// TIA Portal project "projet sadokkkkkkalasou" (V16)
// Vorlageprojekt für das Buch mit Zielsystem S7-1200

(* hardware
DEVICE "S7-1200-Station_1"  S7-1200 Station
   slot 0: "Baugruppenträger_0"  Rack  V1.0
   slot 1: "PLC_1"  CPU 1211C DC/DC/DC  6ES7 211-1AE40-0XB0  V4.1
*)

// ===== PLC "PLC_1"  CPU 1211C DC/DC/DC =====

VAR_GLOBAL   // PLC tag table "Standard-Variablentabelle"
   "km1" AT %Q0.0 : Bool;
   "km2" AT %Q0.2 : Bool;
   "GRAB" AT %Q0.1 : Bool;
   "MOVE X" AT %Q0.3 : Bool;
   "MOVE Z" AT %Q0.4 : Bool;
   "PUSHER" AT %Q0.5 : Bool;
   "LH" AT %I0.1 : Bool;
   "LL" AT %I0.2 : Bool;
   "CP" AT %I0.3 : Bool;
   "CC" AT %I0.4 : Bool;
   "PD" AT %I0.5 : Bool;
   "SZ" AT %I0.6 : Bool;
   "SX" AT %I0.7 : Bool;
   "START" AT %I1.0 : Bool;
   "Moving X" AT %I1.1 : Bool;
   "moving Z" AT %I1.2 : Bool;
   "DS4" AT %I1.3 : Bool;
   "STOP" AT %I1.4 : Bool;
   "km3" AT %Q1.5 : Bool;
   "FC2" AT %I1.6 : Bool;
   "FC1" AT %I1.7 : Bool;
   "Emiteur1" AT %Q2.0 : Bool;
   "Emiteur2" AT %Q2.1 : Bool;
   "Rb1" AT %Q2.2 : Bool;
   "Rb2" AT %Q2.3 : Bool;
   "rs1" AT %I2.4 : Bool;
   "rs2" AT %I2.5 : Bool;
   "cc2" AT %I3.1 : Bool;
   "sz2" AT %I3.2 : Bool;
   "sx2" AT %I3.3 : Bool;
   "rotccw" AT %Q2.4 : Bool;
   "rotcw" AT %Q2.5 : Bool;
   "rot1" AT %I3.4 : Bool;
   "rot4" AT %I2.7 : Bool;
   "km4" AT %Q2.7 : Bool;
   "FC3" AT %I3.0 : Bool;
   "Emiteur3" AT %Q0.6 : Bool;
   "rb3" AT %Q0.7 : Bool;
   "rb31" AT %Q1.0 : Bool;
   "rb32" AT %Q1.1 : Bool;
   "rb11" AT %Q1.2 : Bool;
   "rb21" AT %Q1.3 : Bool;
   "rb22" AT %Q1.4 : Bool;
   "red light" AT %Q1.6 : Bool;
   "green light" AT %Q1.7 : Bool;
   "yellow light" AT %Q2.6 : Bool;
END_VAR

// folder: System blocks/Program resources

DATA_BLOCK "IEC_Timer_0_DB"   // DB1
{ S7_Optimized_Access := 'TRUE' }
AUTHOR : Simatic
FAMILY : IEC
NAME : IEC_TMR
VERSION : 1.0
// stored: InstanceOfName IEC_TIMER
"IEC_TIMER"
BEGIN
END_DATA_BLOCK

DATA_BLOCK "IEC_Timer_0_DB_1"   // DB2
{ S7_Optimized_Access := 'TRUE' }
AUTHOR : Simatic
FAMILY : IEC
NAME : IEC_TMR
VERSION : 1.0
// stored: InstanceOfName IEC_TIMER
"IEC_TIMER"
BEGIN
END_DATA_BLOCK

DATA_BLOCK "IEC_Timer_0_DB_2"   // DB3
{ S7_Optimized_Access := 'TRUE' }
AUTHOR : Simatic
FAMILY : IEC
NAME : IEC_TMR
VERSION : 1.0
// stored: InstanceOfName IEC_TIMER
"IEC_TIMER"
BEGIN
END_DATA_BLOCK

DATA_BLOCK "IEC_Timer_0_DB_3"   // DB4
{ S7_Optimized_Access := 'TRUE' }
AUTHOR : Simatic
FAMILY : IEC
NAME : IEC_TMR
VERSION : 1.0
// stored: InstanceOfName IEC_TIMER
"IEC_TIMER"
BEGIN
END_DATA_BLOCK

DATA_BLOCK "IEC_Timer_0_DB_4"   // DB5
{ S7_Optimized_Access := 'TRUE' }
AUTHOR : Simatic
FAMILY : IEC
NAME : IEC_TMR
VERSION : 1.0
// stored: InstanceOfName IEC_TIMER
"IEC_TIMER"
BEGIN
END_DATA_BLOCK

DATA_BLOCK "IEC_Timer_0_DB_5"   // DB6
{ S7_Optimized_Access := 'TRUE' }
AUTHOR : Simatic
FAMILY : IEC
NAME : IEC_TMR
VERSION : 1.0
// stored: InstanceOfName IEC_TIMER
"IEC_TIMER"
BEGIN
END_DATA_BLOCK

DATA_BLOCK "IEC_Timer_0_DB_8"   // DB7
{ S7_Optimized_Access := 'TRUE' }
AUTHOR : Simatic
FAMILY : IEC
NAME : IEC_TMR
VERSION : 1.0
// stored: InstanceOfName IEC_TIMER
"IEC_TIMER"
BEGIN
END_DATA_BLOCK

DATA_BLOCK "IEC_Timer_0_DB_6"   // DB8
{ S7_Optimized_Access := 'TRUE' }
AUTHOR : Simatic
FAMILY : IEC
NAME : IEC_TMR
VERSION : 1.0
// stored: InstanceOfName IEC_TIMER
"IEC_TIMER"
BEGIN
END_DATA_BLOCK

DATA_BLOCK "IEC_Timer_0_DB_7"   // DB9
{ S7_Optimized_Access := 'TRUE' }
AUTHOR : Simatic
FAMILY : IEC
NAME : IEC_TMR
VERSION : 1.0
// stored: InstanceOfName IEC_TIMER
"IEC_TIMER"
BEGIN
END_DATA_BLOCK

DATA_BLOCK "IEC_Timer_0_DB_9"   // DB10
{ S7_Optimized_Access := 'TRUE' }
AUTHOR : Simatic
FAMILY : IEC
NAME : IEC_TMR
VERSION : 1.0
// stored: InstanceOfName IEC_TIMER
"IEC_TIMER"
BEGIN
END_DATA_BLOCK

DATA_BLOCK "IEC_Timer_0_DB_11"   // DB12
{ S7_Optimized_Access := 'TRUE' }
AUTHOR : Simatic
FAMILY : IEC
NAME : IEC_TMR
VERSION : 1.0
// stored: InstanceOfName IEC_TIMER
"IEC_TIMER"
BEGIN
END_DATA_BLOCK

DATA_BLOCK "IEC_Timer_0_DB_12"   // DB13
{ S7_Optimized_Access := 'TRUE' }
AUTHOR : Simatic
FAMILY : IEC
NAME : IEC_TMR
VERSION : 1.0
// stored: InstanceOfName IEC_TIMER
"IEC_TIMER"
BEGIN
END_DATA_BLOCK

// folder: (top level)

FUNCTION "MHJ-PLC-Lab-Function-S71200" : Void   // FC9000, SCL
{ S7_Optimized_Access := 'TRUE' }
VERSION : 0.1
   VAR_TEMP
      rdTimeReturn : Int;
      outputTime : DTL;
      SyncVal : Byte;
      forVal : Int;
      forVal_2 : Int;
      Value : Byte;
   END_VAR
   VAR CONSTANT
      CompVal : Byte := 16#34;
      Value_01 : Byte := 16#11;
      Value_01_DW : DWord := 16#A165_D992;
      Value_02_DW : DWord := 16#58BE_4401;
   END_VAR
BEGIN

   #Value:=PEEK(area := 16#82,
        dbNumber := 0,
        byteOffset := 511);
   #Value := #Value + 1;

   POKE(area := 16#82,
        dbNumber := 0,
        byteOffset := 511,
        value := #Value);

   POKE(area:=16#81,
        dbNumber:=0,
        byteOffset:=1016,
        value:=#Value_01_DW);
   POKE(area := 16#81,
        dbNumber := 0,
        byteOffset := 1020,
        value := #Value_02_DW);

   POKE(area := 16#81,
        dbNumber := 0,
        byteOffset := 511,
        value := B#16#00);

   FOR #forVal := 0 TO 120 DO
       FOR #forVal_2:=0 TO 10 DO
           #rdTimeReturn:=RD_SYS_T(#outputTime);
           #rdTimeReturn := WR_SYS_T(#outputTime);
           #rdTimeReturn := RD_SYS_T(#outputTime);
           #rdTimeReturn := WR_SYS_T(#outputTime);
       END_FOR;
       #SyncVal:= PEEK(area := 16#81,
                      dbNumber := 0,
                      byteOffset := 511);
       IF #SyncVal = #CompVal THEN
          GOTO M_1;
       END_IF;
   END_FOR;
   RETURN;

   M_1:
   POKE(area := 16#81,
        dbNumber := 0,
        byteOffset := 511,
        value := B#16#0);
END_FUNCTION

ORGANIZATION_BLOCK "Main"   // OB1, LAD, ProgramCycle
TITLE = "Main Program Sweep (Cycle)"
{ S7_Optimized_Access := 'TRUE' }
VERSION : 0.1
   VAR_INPUT
      Initial_Call : Bool;   // Initial call of this OB
      Remanence : Bool;   // =True, if remanent data are available
   END_VAR
   VAR_TEMP   // added for the SCL form of the ladder/FBD networks
      _w1 : Bool;
   END_VAR
BEGIN

REGION Network 1: Konnektierungsbaustein für PLC-Lab / liaison
   // Im Netzwerk 1 wird der Konnektierungsbaustein für PLC-Lab aufgerufen.
   // Dieser Aufruf darf nicht entfernt werden!
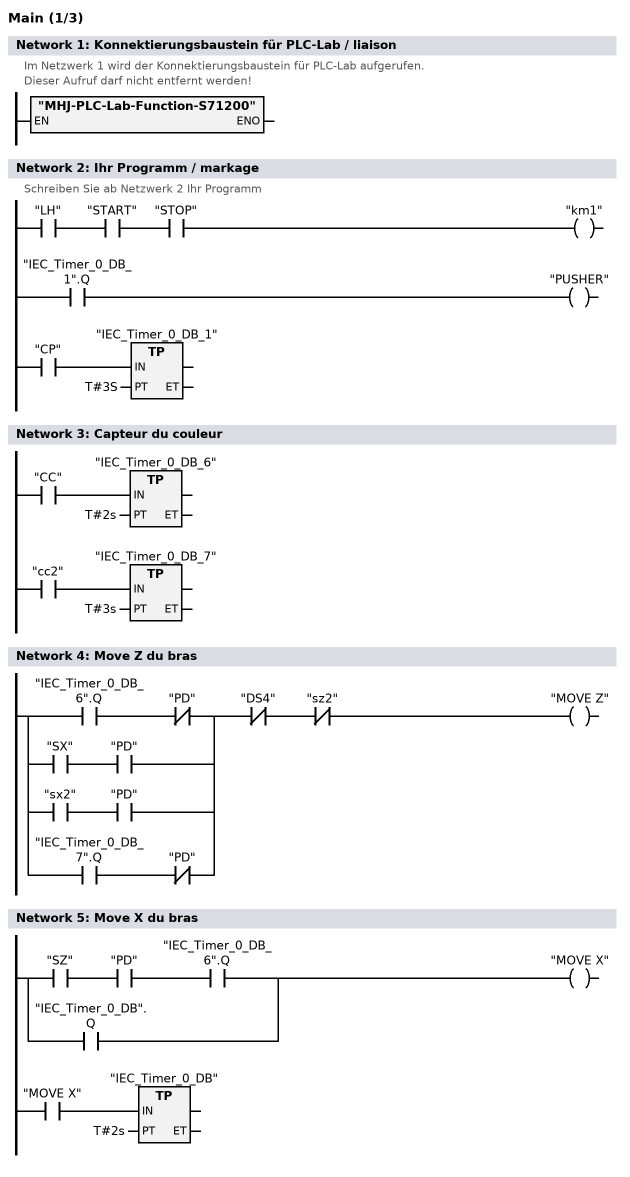
   RUNG wire#powerrail
      "MHJ-PLC-Lab-Function-S71200"()
   END_RUNG
   // the same network as SCL:
   "MHJ-PLC-Lab-Function-S71200"();
END_REGION

REGION Network 2: Ihr Programm / markage
   // Schreiben Sie ab Netzwerk 2 Ihr Programm
   "km1" := "LH" AND "START" AND "STOP";
   "PUSHER" := "IEC_Timer_0_DB_1".Q;
   "IEC_Timer_0_DB_1".TP(IN := "CP", PT := T#3S);
END_REGION

REGION Network 3: Capteur du couleur
   "IEC_Timer_0_DB_6".TP(IN := "CC", PT := T#2s);
   "IEC_Timer_0_DB_7".TP(IN := "cc2", PT := T#3s);
END_REGION

REGION Network 4: Move Z du bras
   RUNG wire#powerrail
      Contact( "IEC_Timer_0_DB_6".Q )
      I_Contact( "PD" )
      wire#w1
      I_Contact( "DS4" )
      I_Contact( "sz2" )
      Coil( "MOVE Z" )
   END_RUNG
   RUNG wire#powerrail
      Contact( "SX" )
      Contact( "PD" )
   END_RUNG wire#w1
   RUNG wire#powerrail
      Contact( "sx2" )
      Contact( "PD" )
   END_RUNG wire#w1
   RUNG wire#powerrail
      Contact( "IEC_Timer_0_DB_7".Q )
      I_Contact( "PD" )
   END_RUNG wire#w1
   // the same network as SCL:
   "MOVE Z" := (("IEC_Timer_0_DB_6".Q AND NOT "PD") OR ("SX" AND "PD") OR ("sx2" AND "PD") OR ("IEC_Timer_0_DB_7".Q AND NOT "PD")) AND NOT "DS4" AND NOT "sz2";
END_REGION

REGION Network 5: Move X du bras
   "MOVE X" := ("SZ" AND "PD" AND "IEC_Timer_0_DB_6".Q) OR "IEC_Timer_0_DB".Q;
   "IEC_Timer_0_DB".TP(IN := "MOVE X", PT := T#2s);
END_REGION

REGION Network 6: Rotation du bras
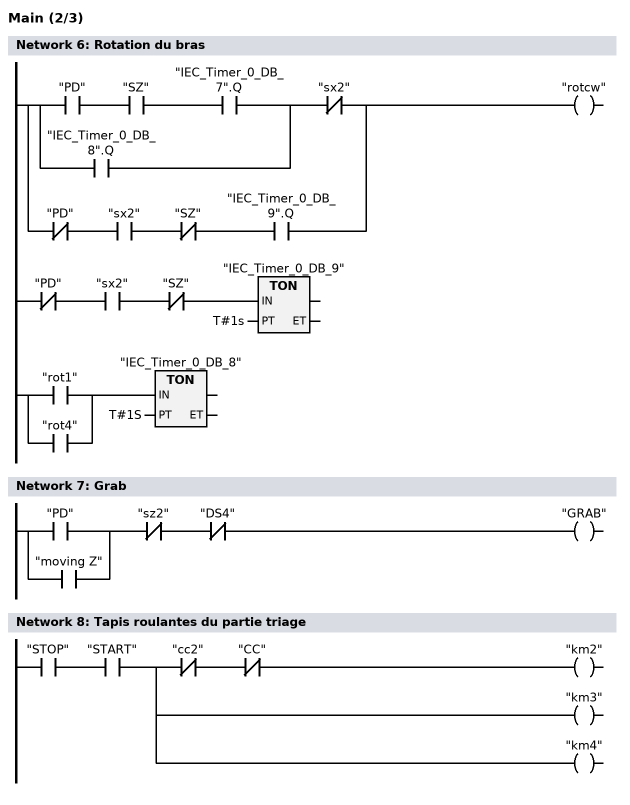
   "rotcw" := ((("PD" AND "SZ" AND "IEC_Timer_0_DB_7".Q) OR "IEC_Timer_0_DB_8".Q) AND NOT "sx2") OR (NOT "PD" AND "sx2" AND NOT "SZ" AND "IEC_Timer_0_DB_9".Q);
   "IEC_Timer_0_DB_9".TON(IN := NOT "PD" AND "sx2" AND NOT "SZ", PT := T#1s);
   "IEC_Timer_0_DB_8".TON(IN := "rot1" OR "rot4", PT := T#1S);
END_REGION

REGION Network 7: Grab
   RUNG wire#powerrail
      Contact( "PD" )
      wire#w1
      I_Contact( "sz2" )
      I_Contact( "DS4" )
      Coil( "GRAB" )
   END_RUNG
   RUNG wire#powerrail
      Contact( "moving Z" )
   END_RUNG wire#w1
   // the same network as SCL:
   "GRAB" := ("PD" OR "moving Z") AND NOT "sz2" AND NOT "DS4";
END_REGION

REGION Network 8: Tapis roulantes du partie triage
   RUNG wire#powerrail
      Contact( "STOP" )
      Contact( "START" )
      wire#w1
      I_Contact( "cc2" )
      I_Contact( "CC" )
      Coil( "km2" )
   END_RUNG
   RUNG wire#w1
      Coil( "km3" )
   END_RUNG
   RUNG wire#w1
      Coil( "km4" )
   END_RUNG
   // the same network as SCL:
   #_w1 := "STOP" AND "START";
   "km2" := #_w1 AND NOT "cc2" AND NOT "CC";
   "km3" := #_w1;
   "km4" := #_w1;
END_REGION

REGION Network 9: Evacuation du piéces
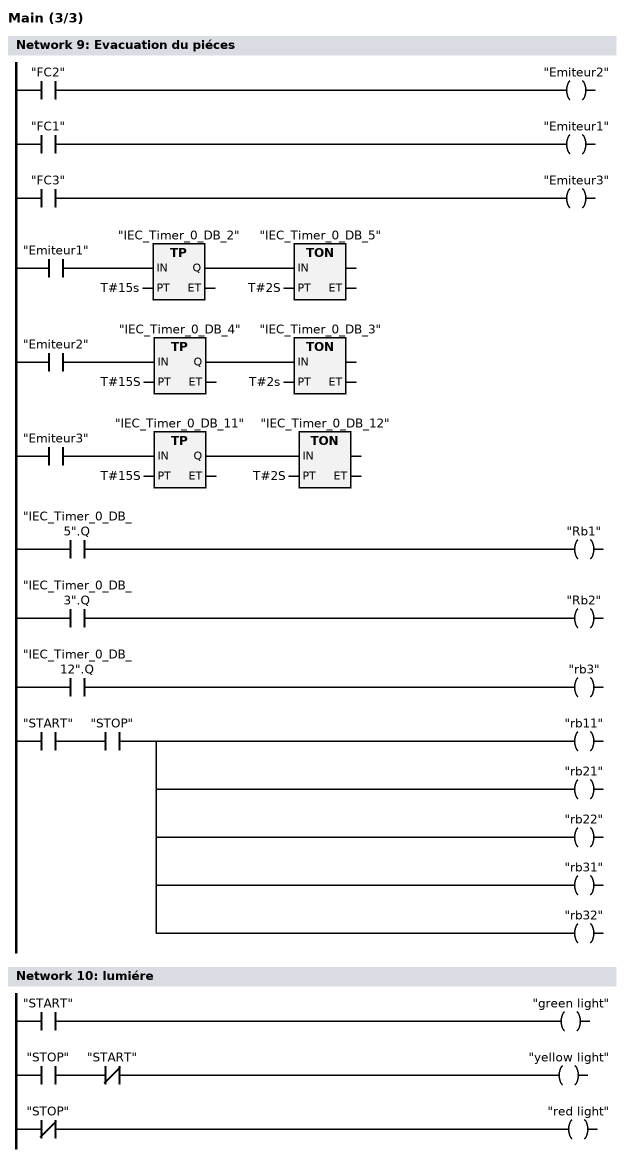
   "Emiteur2" := "FC2";
   "Emiteur1" := "FC1";
   "Emiteur3" := "FC3";
   "IEC_Timer_0_DB_2".TP(IN := "Emiteur1", PT := T#15s);
   "IEC_Timer_0_DB_5".TON(IN := "IEC_Timer_0_DB_2".Q, PT := T#2S);
   "IEC_Timer_0_DB_4".TP(IN := "Emiteur2", PT := T#15S);
   "IEC_Timer_0_DB_3".TON(IN := "IEC_Timer_0_DB_4".Q, PT := T#2s);
   "IEC_Timer_0_DB_11".TP(IN := "Emiteur3", PT := T#15S);
   "IEC_Timer_0_DB_12".TON(IN := "IEC_Timer_0_DB_11".Q, PT := T#2S);
   "Rb1" := "IEC_Timer_0_DB_5".Q;
   "Rb2" := "IEC_Timer_0_DB_3".Q;
   "rb3" := "IEC_Timer_0_DB_12".Q;
   "rb11" := "START" AND "STOP";
   "rb21" := "rb11";
   "rb22" := "rb11";
   "rb31" := "rb11";
   "rb32" := "rb11";
END_REGION

REGION Network 10: lumiére
   RUNG wire#powerrail
      Contact( "START" )
      Coil( "green light" )
   END_RUNG
   RUNG wire#powerrail
      Contact( "STOP" )
      I_Contact( "START" )
      Coil( "yellow light" )
   END_RUNG
   RUNG wire#powerrail
      I_Contact( "STOP" )
      Coil( "red light" )
   END_RUNG
   // the same network as SCL:
   "green light" := "START";
   "yellow light" := "STOP" AND NOT "START";
   "red light" := NOT "STOP";
END_REGION
END_ORGANIZATION_BLOCK